TYPE "EM_Carriage_Pendant_State"
VERSION : 0.1
   STRUCT
      state : Int;
      step : Int;
      done : Bool;
      fault : Bool;
   END_STRUCT;
END_TYPE
